(* CoDeSys 2.3.8.1 project: OPC_Test.pro *)
(* Libraries: Standard.lib 4.10.05 11:14:46, IecSfc.lib 13.4.06 15:51:28, SYSLIBCALLBACK.LIB 16.4.07 16:52:46 *)

(* POU PLC_PRG, ST *)
PROGRAM PLC_PRG
VAR
	blVar: BOOL;
	shortVal: SINT;
	intVal: INT;
	dintVal: DINT;
	uintVal: UINT;
	udintVal: UDINT;
	floatVal: REAL;
	doubleVal: LREAL;
	oneSecT: TON;
END_VAR
oneSecT(IN := NOT oneSecT.Q, PT:= t#2s);

IF(oneSecT.Q) THEN
	blVar := NOT blVar;
	shortVal := shortVal + 1;
	intVal := intVal + 5;
	dintVal := dintVal + 15;
	uintVal := uintVal + 8;
	udintVal := udintVal + 149;
	floatVal := floatVal + 1.58;
	doubleVal := doubleVal + 89.754;
END_IF;

IF(shortVal > 100) THEN shortVal := 0; END_IF;
IF(intVal > 32000) THEN intVal := 0; END_IF;
IF(dintVal > 1000000) THEN dintVal := 0; END_IF;
IF(uintVal > 60000) THEN uintVal := 0; END_IF;
IF(udintVal > 6000000) THEN udintVal := 0; END_IF;
IF(floatVal > 100.0) THEN floatVal := 0; END_IF;
IF(doubleVal > 100000.0) THEN doubleVal := 0; END_IF;
END_PROGRAM
